FUNCTION toggleIntermediateCircuitPump : BOOL
VAR_INPUT
	pMachine : POINTER TO FB_StateMachine;
END_VAR
VAR
END_VAR

// Das manuelle Ein-Ausschalten der Zwischenkreispumpe ist nur in IDLE oder ERROR Status möglich
IF pMachine^.iState.State = E_State.IDLE OR pMachine^.iState.State = E_State.ERROR THEN
	IF pMachine^.pd.actor.operatingStateIntermediateCircuitPump = FALSE THEN
		LogMessage(E_LogType.INFO, 'Schalte Sole Zwischenkreispumpe: -> ', 'Ein');	
		pMachine^.pd.actor.operatingStateIntermediateCircuitPump := TRUE;
	ELSE
		LogMessage(E_LogType.INFO, 'Schalte Sole Zwischenkreispumpe: -> ', 'Aus');	
		pMachine^.pd.actor.operatingStateIntermediateCircuitPump := FALSE;
	END_IF
END_IF

END_FUNCTION

(* stored: Version 1.1.0.1
   POU toggleIntermediateCircuitPump: Id {a179cbaa-be08-4b5d-863d-d11cdf9bb358}, SpecialFunc None *)
